(* Logix 5000 project; controller test vendor 1 type 14 code 151 rev 32.13; software revision 32.02; part 3 of 4 *)
(* tags used below, declared in another part *)
   _CopDes1 : DINT;
   _CopDes4 : DINT;
   _CopDes5 : DINT;
   _CopDes6 : DINT;
   _CopDes8 : DINT;
   _CopLength : DINT;
   _CopLength1 : DINT;
   _CopLength3 : DINT;
   _CopLength4 : DINT;
   _CopLength5 : DINT;
   _CopLength6 : DINT;
   _CopLength7 : DINT;
   _CopLength8 : DINT;
   _CopSource : DINT;
   _CopSource1 : DINT;
   _CopSource3 : DINT;
   _CopSource4 : DINT;
   _CopSource5 : DINT;
   _CopSource6 : DINT;
   _CopSource7 : DINT;
   _CopSource8 : DINT;
   _edbAoiFilterFlowAir : AOI_FilterSignal;
   _edbAoiFilterFlowO2 : AOI_FilterSignal;
   _edbAoiFilterPress : AOI_FilterSignal;
   _edbCanStore : BOOL;
   _edbFlowArrFiltered : REAL[1000,2];
   _edbFlowO2Filtered : REAL[1000,2];
   _edbHalfWindowFilterSize : DINT;
   _edbIdx : DINT;
   _edbParUseWeigths : BOOL;
   _edbParWeights : REAL[31];
   _edbPressArrFiltered : REAL[1000,2];
   _edbTypeOfFilter : DINT;
   _endPosition : DINT;
   _endPositionOld : DINT;
   _EndSendPosition : DINT;
   _i : DINT;
   _PointAfterEnd : DINT;
   _StartPointBerfore : DINT;
   _StartPosition : DINT;
   _StartpositionOld : DINT;
   AirConstantFlow : REAL;
   AirmADer : REAL;
   AirmAOut : REAL;
   AirmASlope : REAL;
   AirRampFlowIncreasePerAdjust : REAL;
   AirUp : CAM_PROFILE[1010];
   AnalogInputFlow : ALIAS FOR Local:2:I.Ch3Data;
   AnalogInputFlowAir : ALIAS FOR Local:2:I.Ch1Data;
   AnalogInputFlowO2 : ALIAS FOR Local:2:I.Ch0Data;
   AnalogInputPressure : ALIAS FOR Local:2:I.Ch2Data;
   AnalogOutFlowAir : ALIAS FOR Local:2:O.Ch1Data;
   AnalogOutFlowO2 : ALIAS FOR Local:2:O.Ch0Data;
   BreathDetect : BOOL;
   BreathDurationArr : REAL[50];   // 50 length array with seconds for each breath for calculation of minute avgVentStateArr. Calcualted from knowing meas at
   BreathDurationInMS : REAL;
   CalcNewData : BOOL;
   ConstansFlowNrCalc : REAL;
   ConstantFlowNrOfAdjustments : REAL;
   ConstantFlowTimeInMS : REAL;
   ConstantInspiratoryFlow : REAL;
   counter : DINT;   // Counter for Flow fill array
   CrsDynArr : REAL[50];   // 50 length array with dynamic respiraotry system compliance in ml/cmH2O, from measCalc()
   CrsQStatArr : REAL[50];   // 50 length array with quasistatic respiratory system compliance in ml/cmH2O, from measCalc()
   CsumData : DINT;
   CsumDataOld : DINT;
   data_changed : BOOL;
   endI : DINT;
   Exp : BOOL;
   expCount : INT;   // between 1-1000 to indicate where valveCtrl should read from expOpenCloseCtrl[]
   expCountLength : INT;   // between 1-1000 to indicate when valveCtrl should stop reading from expOpenCloseCtrl[], copied from nextExpCountLength by
   expCountlengthCalc : REAL;
   expCountLengthNew : REAL;
   expEndI : INT;
   expOpen : ALIAS FOR Local:1:O.Data.0;
   expOpenCloseCtrl : INT[1000];   // 1000 length array with open (1) or close (0) for exp valve, moved from nextexpOpenCloseCtrl[] by ISR_ValveCtrl()
   expOpenCloseCtrlNew : INT[1000];
   expStartI : INT;
   expTimeInMS : REAL;
   F1_pushed_new : BOOL;
   F1_pushed_old : BOOL;
   F2_pushed_new : BOOL;
   F2_pushed_old : BOOL;
   F3_pushed_new : BOOL;
   F3_pushed_old : BOOL;
   Fill : AOI_FillArrayReal;
   Fill50 : AOI_FillArrayReal50;
   Fillint : AOI_FillArrayInt;
   FillLoop : AOI_FillArray_Real2D;
   FiO2 : INT;   // 25-100%
   FiO2Running : INT;
   Floor : AOI_Floor;
   FlowAir : REAL[1000,2];   // 1000 length 2D FIFO array with flow values and status bits indicating if values have been analysed (1) or not (0) by mea
   FlowArrMem : REAL[1000,2];
   flowCalcOn : BOOL;
   FlowImaxArr : REAL[50];   // 50 length array with max insp flow in l/min, from measCalc()
   FlowO2 : REAL[1000,2];
   FlowO2Mem : REAL[1000,2];
   FractionAir : REAL;
   FractionO2 : REAL;
   GetSlaveValue : MOTION_INSTRUCTION;
   HMI_ScreenNo : DINT;
   HMIStart : BOOL;
   HMIStop : BOOL;
   i : DINT;
   I_E : STRING;   // part of I:E ratio: 1, 2, 3 or 4
   IE : STRING[4];
   IE_counter : DINT;
   IE_E : INT;
   IE_ERunning : INT;
   IE_I : INT;
   IE_IRunning : INT;
   Insp : BOOL;
   inspAirFlowCtrl : REAL[650];   // 650 length array with flow values for insp air valve, moved from nextInspAirFlowCtrl[] by ISR_ValveCtrl()
   inspAirFlowCtrlNew : REAL[650];
   inspCount : INT;   // between 1-650 to indicate where valveCtrl should read from inspAirFlowCtrl[] and inspO2FlowCtrl[]
   inspCountLength : INT;   // between 1-650 to indicate when valveCtrl should stop reading from inspAirFlowCtrl[] and inspO2FlowCtrl[], copied from ne
   inspCountLengthNew : REAL;
   inspCounts : REAL;
   InspiratoryRampTimeInMS : REAL;
   inspO2FlowCtrl : REAL[650];   // 650 length array with flow values for insp O2 valve, moved from nextInspO2FlowCtrl[] by ISR_ValveCtrl()
   inspO2FlowCtrlNew : REAL[650];
   inspPauseCalc : REAL;
   inspPauseNrOfAdjustments : REAL;
   inspPauseStartI : INT;
   inspPauseTime : INT;
   inspPauseTimeInMS : REAL;
   inspPauseTimePercent : REAL;
   inspPauseTimeRunning : INT;
   inspRampTime : INT;
   inspRampTimePercent : REAL;
   inspRampTimeRunning : INT;
   inspStartI : INT;
   inspTimeinMS : REAL;
   last_state : DINT;
   maxFlowAllowed : INT;
   message : STRING;
   Messages_to_user : STRING[10];
   Mode : STRING;
   MVArr : REAL[50];   // 50 length array with minute ventilation in l/min, from measCalc()
   NewExpOpenCloseAvail : BOOL;   // signal to valveCtrl to include new expOpenCloseCtrl[]to overwrite when expiration ended, set by calcBreath()
   newInspFlowAvil : BOOL;
   NewSettings : BOOL;
   NewTimeRate_p5 : DINT;
   NewTimeRate_p8 : DINT;
   nextExpCountLength : INT;   // between 1-1000 to indicate when valveCtrl should stop reading from expOpenCloseCtrl[], set by calcBreath()
   nextExpOpenCloseCtrl : INT[1000];   // 1000 length array with open (1) or close (0) for exp valve, set by calcBreath()
   nextInspAirFlowCtrl : REAL[650];   // 650 length array with flow values for insp air valve, set by calcBreath()
   nextInspCountLength : INT;   // between 1-650 to indicate when valveCtrl should stop reading from inspAirFlowCtrl[] and inspO2FlowCtrl[], set by calcBre
   nextInspO2FlowCtrl : REAL[650];   // 650 length array with flow values for insp O2 valve, set by calcBreath()
   O2 : DINT;
   O2ConstantFlow : REAL;
   O2mADer : REAL;
   O2mAOut : REAL;
   O2mASlope : REAL;
   O2RampFlowIncreasePerAdjust : REAL;
   O2Up : CAM_PROFILE[1010];

        [540].Status := 2, [541].Status := 2, [542].Status := 2, [543].Status := 2, [544].Status := 2, [545].Status := 2, [546].Status := 2, [547].Status := 2, [548].Status := 2, [549].Status := 2, [550].Status := 2, [551].Status := 2, [552].Status := 2, [553].Status := 2, [554].Status := 2, [555].Status := 2, [556].Status := 2, [557].Status := 2, [558].Status := 2, [559].Status := 2, [560].Status := 2, [561].Status := 2, [562].Status := 2, [563].Status := 2, [564].Status := 2, [565].Status := 2, [566].Status := 2, [567].Status := 2, [568].Status := 2, [569].Status := 2, [570].Status := 2, [571].Status := 2, [572].Status := 2, [573].Status := 2, [574].Status := 2, [575].Status := 2, [576].Status := 2, [577].Status := 2, [578].Status := 2, [579].Status := 2, [580].Status := 2, [581].Status := 2, [582].Status := 2, [583].Status := 2, [584].Status := 2, [585].Status := 2, [586].Status := 2, [587].Status := 2, [588].Status := 2, [589].Status := 2, [590].Status := 2, [591].Status := 2, [592].Status := 2, [593].Status := 2, [594].Status := 2, [595].Status := 2, [596].Status := 2, [597].Status := 2, [598].Status := 2, [599].Status := 2,
        [600].Status := 2, [601].Status := 2, [602].Status := 2, [603].Status := 2, [604].Status := 2, [605].Status := 2, [606].Status := 2, [607].Status := 2, [608].Status := 2, [609].Status := 2, [610].Status := 2, [611].Status := 2, [612].Status := 2, [613].Status := 2, [614].Status := 2, [615].Status := 2, [616].Status := 2, [617].Status := 2, [618].Status := 2, [619].Status := 2, [620].Status := 2, [621].Status := 2, [622].Status := 2, [623].Status := 2, [624].Status := 2, [625].Status := 2, [626].Status := 2, [627].Status := 2, [628].Status := 2, [629].Status := 2, [630].Status := 2, [631].Status := 2, [632].Status := 2, [633].Status := 2, [634].Status := 2, [635].Status := 2, [636].Status := 2, [637].Status := 2, [638].Status := 2, [639].Status := 2, [640].Status := 2, [641].Status := 2, [642].Status := 2, [643].Status := 2, [644].Status := 2, [645].Status := 2, [646].Status := 2, [647].Status := 2, [648].Status := 2, [649].Status := 2, [650].Status := 2, [651].Status := 2, [652].Status := 2, [653].Status := 2, [654].Status := 2, [655].Status := 2, [656].Status := 2, [657].Status := 2, [658].Status := 2, [659].Status := 2,
        [660].Status := 2, [661].Status := 2, [662].Status := 2, [663].Status := 2, [664].Status := 2, [665].Status := 2, [666].Status := 2, [667].Status := 2, [668].Status := 2, [669].Status := 2, [670].Status := 2, [671].Status := 2, [672].Status := 2, [673].Status := 2, [674].Status := 2, [675].Status := 2, [676].Status := 2, [677].Status := 2, [678].Status := 2, [679].Status := 2, [680].Status := 2, [681].Status := 2, [682].Status := 2, [683].Status := 2, [684].Status := 2, [685].Status := 2, [686].Status := 2, [687].Status := 2, [688].Status := 2, [689].Status := 2, [690].Status := 2, [691].Status := 2, [692].Status := 2, [693].Status := 2, [694].Status := 2, [695].Status := 2, [696].Status := 2, [697].Status := 2, [698].Status := 2, [699].Status := 2, [700].Status := 2, [701].Status := 2, [702].Status := 2, [703].Status := 2, [704].Status := 2, [705].Status := 2, [706].Status := 2, [707].Status := 2, [708].Status := 2, [709].Status := 2, [710].Status := 2, [711].Status := 2, [712].Status := 2, [713].Status := 2, [714].Status := 2, [715].Status := 2, [716].Status := 2, [717].Status := 2, [718].Status := 2, [719].Status := 2,
        [720].Status := 2, [721].Status := 2, [722].Status := 2, [723].Status := 2, [724].Status := 2, [725].Status := 2, [726].Status := 2, [727].Status := 2, [728].Status := 2, [729].Status := 2, [730].Status := 2, [731].Status := 2, [732].Status := 2, [733].Status := 2, [734].Status := 2, [735].Status := 2, [736].Status := 2, [737].Status := 2, [738].Status := 2, [739].Status := 2, [740].Status := 2, [741].Status := 2, [742].Status := 2, [743].Status := 2, [744].Status := 2, [745].Status := 2, [746].Status := 2, [747].Status := 2, [748].Status := 2, [749].Status := 2, [750].Status := 2, [751].Status := 2, [752].Status := 2, [753].Status := 2, [754].Status := 2, [755].Status := 2, [756].Status := 2, [757].Status := 2, [758].Status := 2, [759].Status := 2, [760].Status := 2, [761].Status := 2, [762].Status := 2, [763].Status := 2, [764].Status := 2, [765].Status := 2, [766].Status := 2, [767].Status := 2, [768].Status := 2, [769].Status := 2, [770].Status := 2, [771].Status := 2, [772].Status := 2, [773].Status := 2, [774].Status := 2, [775].Status := 2, [776].Status := 2, [777].Status := 2, [778].Status := 2, [779].Status := 2,
        [780].Status := 2, [781].Status := 2, [782].Status := 2, [783].Status := 2, [784].Status := 2, [785].Status := 2, [786].Status := 2, [787].Status := 2, [788].Status := 2, [789].Status := 2, [790].Status := 2, [791].Status := 2, [792].Status := 2, [793].Status := 2, [794].Status := 2, [795].Status := 2, [796].Status := 2, [797].Status := 2, [798].Status := 2, [799].Status := 2, [800].Status := 2, [801].Status := 2, [802].Status := 2, [803].Status := 2, [804].Status := 2, [805].Status := 2, [806].Status := 2, [807].Status := 2, [808].Status := 2, [809].Status := 2, [810].Status := 2, [811].Status := 2, [812].Status := 2, [813].Status := 2, [814].Status := 2, [815].Status := 2, [816].Status := 2, [817].Status := 2, [818].Status := 2, [819].Status := 2, [820].Status := 2, [821].Status := 2, [822].Status := 2, [823].Status := 2, [824].Status := 2, [825].Status := 2, [826].Status := 2, [827].Status := 2, [828].Status := 2, [829].Status := 2, [830].Status := 2, [831].Status := 2, [832].Status := 2, [833].Status := 2, [834].Status := 2, [835].Status := 2, [836].Status := 2, [837].Status := 2, [838].Status := 2, [839].Status := 2,
        [840].Status := 2, [841].Status := 2, [842].Status := 2, [843].Status := 2, [844].Status := 2, [845].Status := 2, [846].Status := 2, [847].Status := 2, [848].Status := 2, [849].Status := 2, [850].Status := 2, [851].Status := 2, [852].Status := 2, [853].Status := 2, [854].Status := 2, [855].Status := 2, [856].Status := 2, [857].Status := 2, [858].Status := 2, [859].Status := 2, [860].Status := 2, [861].Status := 2, [862].Status := 2, [863].Status := 2, [864].Status := 2, [865].Status := 2, [866].Status := 2, [867].Status := 2, [868].Status := 2, [869].Status := 2, [870].Status := 2, [871].Status := 2, [872].Status := 2, [873].Status := 2, [874].Status := 2, [875].Status := 2, [876].Status := 2, [877].Status := 2, [878].Status := 2, [879].Status := 2, [880].Status := 2, [881].Status := 2, [882].Status := 2, [883].Status := 2, [884].Status := 2, [885].Status := 2, [886].Status := 2, [887].Status := 2, [888].Status := 2, [889].Status := 2, [890].Status := 2, [891].Status := 2, [892].Status := 2, [893].Status := 2, [894].Status := 2, [895].Status := 2, [896].Status := 2, [897].Status := 2, [898].Status := 2, [899].Status := 2,
        [900].Status := 2, [901].Status := 2, [902].Status := 2, [903].Status := 2, [904].Status := 2, [905].Status := 2, [906].Status := 2, [907].Status := 2, [908].Status := 2, [909].Status := 2, [910].Status := 2, [911].Status := 2, [912].Status := 2, [913].Status := 2, [914].Status := 2, [915].Status := 2, [916].Status := 2, [917].Status := 2, [918].Status := 2, [919].Status := 2, [920].Status := 2, [921].Status := 2, [922].Status := 2, [923].Status := 2, [924].Status := 2, [925].Status := 2, [926].Status := 2, [927].Status := 2, [928].Status := 2, [929].Status := 2, [930].Status := 2, [931].Status := 2, [932].Status := 2, [933].Status := 2, [934].Status := 2, [935].Status := 2, [936].Status := 2, [937].Status := 2, [938].Status := 2, [939].Status := 2, [940].Status := 2, [941].Status := 2, [942].Status := 2, [943].Status := 2, [944].Status := 2, [945].Status := 2, [946].Status := 2, [947].Status := 2, [948].Status := 2, [949].Status := 2, [950].Status := 2, [951].Status := 2, [952].Status := 2, [953].Status := 2, [954].Status := 2, [955].Status := 2, [956].Status := 2, [957].Status := 2, [958].Status := 2, [959].Status := 2,
        [960].Status := 2, [961].Status := 2, [962].Status := 2, [963].Status := 2, [964].Status := 2, [965].Status := 2, [966].Status := 2, [967].Status := 2, [968].Status := 2, [969].Status := 2, [970].Status := 2, [971].Status := 2, [972].Status := 2, [973].Status := 2, [974].Status := 2, [975].Status := 2, [976].Status := 2, [977].Status := 2, [978].Status := 2, [979].Status := 2, [980].Status := 2, [981].Status := 2, [982].Status := 2, [983].Status := 2, [984].Status := 2, [985].Status := 2, [986].Status := 2, [987].Status := 2, [988].Status := 2, [989].Status := 2, [990].Status := 2, [991].Status := 2, [992].Status := 2, [993].Status := 2, [994].Status := 2, [995].Status := 2, [996].Status := 2, [997].Status := 2, [998].Status := 2, [999].Status := 2, [1000].Status := 2, [1001].Status := 2, [1002].Status := 2);
   PEEP : REAL := 4402.0;   // positive end expiratory pressure in cmH2O
   PEEPArr : REAL[50];   // 50 length array with positive end expiratory pressure in cmH2O, from measCalc()
   PEEPi : REAL;
   PEEPiArr : REAL[50];
   Ppeak : REAL := 10534.0;   // Ppeak
   PpeakArr : REAL[50];   // 50 length array with Ppeak from measCalc(), used for minAvg
   PpeakMaxValue : AOI_Max := (Out_Max := 10534.0, _i := 196);
   Pplat : REAL := 9761.556;   // plateau insp pressure in cmH2O
   PplatArr : REAL[50];   // 50 length array with plateau insp pressure in cmH2O, from measCalc()
   PplatBreathFrac : REAL := 0.2;
   PplatMean : AOI_Mean2D := (In_N0 := 186, In_N1 := 194, Out_Mean := 9761.556, _i := 195);
   PressArr : REAL[1000,2] := ([0,0] := 24.938433, [1,0] := 24.938433, [2,0] := 25.22523, [3,0] := 25.22523, [4,0] := 25.22523, [5,0] := 25.429173, [6,0] := 25.429173, [7,0] := 25.129631, [8,0] := 25.129631, [9,0] := 25.129631, [10,0] := 25.161495, [11,0] := 25.161495, [12,0] := 25.034033, [13,0] := 25.034033, [14,0] := 25.174244, [15,0] := 25.174244, [16,0] := 25.174244, [17,0] := 25.429173, [18,0] := 25.429173, [19,0] := 25.193363, [20,0] := 25.193363, [21,0] := 25.193363, [22,0] := 25.180616, [23,0] := 25.180616, [24,0] := 25.002167, [25,0] := 25.002167, [26,0] := 25.002167, [27,0] := 25.10414, [28,0] := 25.10414, [29,0] := 25.461039, [30,0] := 25.461039, [31,0] := 25.218855, [32,0] := 25.218855, [33,0] := 25.218855, [34,0] := 25.161495, [35,0] := 25.161495, [36,0] := 25.040407, [37,0] := 25.040407, [38,0] := 25.040407, [39,0] := 25.24435, [40,0] := 25.24435, [41,0] := 25.499277, [42,0] := 25.499277, [43,0] := 25.142378, [44,0] := 25.142378, [45,0] := 25.142378, [46,0] := 24.925688, [47,0] := 24.925688, [48,0] := 25.199736, [49,0] := 25.199736, [50,0] := 25.199736, [51,0] := 25.237976, [52,0] := 25.237976, [53,0] := 25.378187, [54,0] := 25.378187, [55,0] := 25.136003, [56,0] := 25.136003, [57,0] := 25.136003, [58,0] := 24.976673, [59,0] := 24.976673,
        [60,0] := 25.199736, [61,0] := 25.199736, [62,0] := 25.199736, [63,0] := 25.136003, [64,0] := 25.136003, [65,0] := 25.403679, [66,0] := 25.403679, [67,0] := 25.212482, [68,0] := 25.212482, [69,0] := 25.212482, [70,0] := 24.906569, [71,0] := 24.906569, [72,0] := 25.212482, [73,0] := 25.212482, [74,0] := 25.212482, [75,0] := 25.269842, [76,0] := 25.269842, [77,0] := 25.359066, [78,0] := 25.359066, [79,0] := 25.359066, [80,0] := 25.193363, [81,0] := 25.193363, [82,0] := 24.912941, [83,0] := 24.912941, [84,0] := 25.250723, [85,0] := 25.250723, [86,0] := 25.250723, [87,0] := 25.282587, [88,0] := 25.282587, [89,0] := 25.308083, [90,0] := 25.308083, [91,0] := 25.116884, [92,0] := 25.116884, [93,0] := 25.116884, [94,0] := 24.925688, [95,0] := 24.925688, [96,0] := 25.20611, [97,0] := 25.20611, [98,0] := 25.20611, [99,0] := 25.250723, [100,0] := 25.250723, [101,0] := 25.314455, [102,0] := 25.314455, [103,0] := 25.193363, [104,0] := 25.193363, [105,0] := 25.193363, [106,0] := 24.938433, [107,0] := 24.938433, [108,0] := 25.193363, [109,0] := 25.193363, [110,0] := 25.193363, [111,0] := 25.308083, [112,0] := 25.308083, [113,0] := 25.276215, [114,0] := 25.276215, [115,0] := 25.276215, [116,0] := 25.193363, [117,0] := 25.193363, [118,0] := 24.93206, [119,0] := 24.93206,
        [120,0] := 25.174244, [121,0] := 25.174244, [122,0] := 25.174244, [123,0] := 25.518398, [124,0] := 25.518398, [125,0] := 25.180616, [126,0] := 25.180616, [127,0] := 25.180616, [128,0] := 25.193363, [129,0] := 25.193363, [130,0] := 25.021286, [131,0] := 25.021286, [132,0] := 25.22523, [133,0] := 25.22523, [134,0] := 25.22523, [135,0] := 25.473785, [136,0] := 25.473785, [137,0] := 25.167871, [138,0] := 25.167871, [139,0] := 25.167871, [140,0] := 25.199736, [141,0] := 25.199736, [142,0] := 25.014912, [143,0] := 25.014912, [144,0] := 25.014912, [145,0] := 25.136003, [146,0] := 25.136003, [147,0] := 25.461039, [148,0] := 25.461039, [149,0] := 25.167871, [150,0] := 25.167871, [151,0] := 25.167871, [152,0] := 25.199736, [153,0] := 25.199736, [154,0] := 25.027658, [155,0] := 25.027658, [156,0] := 25.180616, [157,0] := 25.180616, [158,0] := 25.180616, [159,0] := 25.52477, [160,0] := 25.52477, [161,0] := 25.199736, [162,0] := 25.199736, [163,0] := 25.199736, [164,0] := 25.00854, [165,0] := 25.00854, [166,0] := 25.116884, [167,0] := 25.116884, [168,0] := 25.116884, [169,0] := 25.231602, [170,0] := 25.231602, [171,0] := 25.416426, [172,0] := 25.416426, [173,0] := 25.136003, [174,0] := 25.136003, [175,0] := 25.136003, [176,0] := 24.9703, [177,0] := 24.9703, [178,0] := 25.212482, [179,0] := 25.212482,
        [180,0] := 25.212482, [181,0] := 25.161495, [182,0] := 25.161495, [183,0] := 25.410053, [184,0] := 25.410053, [185,0] := 25.18699, [186,0] := 25.18699, [187,0] := 25.18699, [188,0] := 24.9703, [189,0] := 24.9703, [190,0] := 25.14875, [191,0] := 25.14875, [192,0] := 25.14875, [193,0] := 25.155123, [194,0] := 25.155123, [195,0] := 25.448294, [196,0] := 25.448294, [197,0] := 25.167871, [198,0] := 25.167871, [199,0] := 25.167871, [200,0] := 24.855581, [201,0] := 24.855581, [202,0] := 25.123259, [203,0] := 25.123259, [204,0] := 25.123259, [205,0] := 25.250723, [206,0] := 25.250723, [207,0] := 25.352694, [208,0] := 25.352694, [209,0] := 25.110512, [210,0] := 25.110512, [211,0] := 25.110512, [212,0] := 24.944807, [213,0] := 24.944807, [214,0] := 25.231602, [215,0] := 25.231602, [216,0] := 25.231602, [217,0] := 25.180616, [218,0] := 25.180616, [219,0] := 25.257095, [220,0] := 25.257095, [221,0] := 25.257095, [222,0] := 25.155123, [223,0] := 25.155123, [224,0] := 24.9703, [225,0] := 24.9703, [226,0] := 25.167871, [227,0] := 25.167871, [228,0] := 25.167871, [229,0] := 25.276215, [230,0] := 25.276215, [231,0] := 25.24435, [232,0] := 25.24435, [233,0] := 25.199736, [234,0] := 25.199736, [235,0] := 25.199736, [236,0] := 24.855581, [237,0] := 24.855581, [238,0] := 25.167871, [239,0] := 25.167871,
        [240,0] := 25.167871, [241,0] := 25.38456, [242,0] := 25.38456, [243,0] := 25.250723, [244,0] := 25.250723, [245,0] := 25.250723, [246,0] := 25.155123, [247,0] := 25.155123, [248,0] := 24.900196, [249,0] := 24.900196, [250,0] := 25.237976, [251,0] := 25.237976, [252,0] := 25.237976, [253,0] := 25.461039, [254,0] := 25.461039, [255,0] := 25.193363, [256,0] := 25.193363, [257,0] := 25.193363, [258,0] := 25.199736, [259,0] := 25.199736, [260,0] := 25.00854, [261,0] := 25.00854, [262,0] := 25.237976, [263,0] := 25.237976, [264,0] := 25.237976, [265,0] := 25.422798, [266,0] := 25.422798, [267,0] := 25.193363, [268,0] := 25.193363, [269,0] := 25.193363, [270,0] := 25.18699, [271,0] := 25.18699, [272,0] := 25.065899, [273,0] := 25.065899, [274,0] := 25.155123, [275,0] := 25.155123, [276,0] := 25.155123, [277,0] := 25.473785, [278,0] := 25.473785, [279,0] := 25.20611, [280,0] := 25.20611, [281,0] := 25.20611, [282,0] := 24.98942, [283,0] := 24.98942, [284,0] := 25.142378, [285,0] := 25.142378, [286,0] := 25.142378, [287,0] := 25.250723, [288,0] := 25.250723, [289,0] := 25.48653, [290,0] := 25.48653, [291,0] := 25.142378, [292,0] := 25.142378, [293,0] := 25.142378, [294,0] := 24.893822, [295,0] := 24.893822, [296,0] := 25.199736, [297,0] := 25.199736, [298,0] := 25.199736, [299,0] := 25.193363,
        [300,0] := 25.193363, [301,0] := 25.295334, [302,0] := 25.295334, [303,0] := 25.199736, [304,0] := 25.199736, [305,0] := 25.199736, [306,0] := 24.944807, [307,0] := 24.944807, [308,0] := 25.193363, [309,0] := 25.193363, [310,0] := 25.193363, [311,0] := 25.212482, [312,0] := 25.212482, [313,0] := 25.371813, [314,0] := 25.371813, [315,0] := 25.371813, [316,0] := 25.250723, [317,0] := 25.250723, [318,0] := 24.8747, [319,0] := 24.8747, [320,0] := 25.167871, [321,0] := 25.167871, [322,0] := 25.167871, [323,0] := 25.269842, [324,0] := 25.269842, [325,0] := 25.36544, [326,0] := 25.36544, [327,0] := 25.180616, [328,0] := 25.180616, [329,0] := 25.180616, [330,0] := 24.849209, [331,0] := 24.849209, [332,0] := 25.199736, [333,0] := 25.199736, [334,0] := 25.199736, [335,0] := 25.333574, [336,0] := 25.333574, [337,0] := 25.250723, [338,0] := 25.250723, [339,0] := 25.250723, [340,0] := 25.123259, [341,0] := 25.123259, [342,0] := 24.893822, [343,0] := 24.893822, [344,0] := 25.22523, [345,0] := 25.22523, [346,0] := 25.22523, [347,0] := 25.346321, [348,0] := 25.346321, [349,0] := 25.199736, [350,0] := 25.199736, [351,0] := 25.199736, [352,0] := 25.212482, [353,0] := 25.212482, [354,0] := 25.002167, [355,0] := 25.002167, [356,0] := 25.212482, [357,0] := 25.212482, [358,0] := 25.212482, [359,0] := 25.480158,
        [360,0] := 25.480158, [361,0] := 25.24435, [362,0] := 25.24435, [363,0] := 25.24435, [364,0] := 25.161495, [365,0] := 25.161495, [366,0] := 25.014912, [367,0] := 25.014912, [368,0] := 25.218855, [369,0] := 25.218855, [370,0] := 25.218855, [371,0] := 25.52477, [372,0] := 25.52477, [373,0] := 25.218855, [374,0] := 25.218855, [375,0] := 25.218855, [376,0] := 25.167871, [377,0] := 25.167871, [378,0] := 25.065899, [379,0] := 25.065899, [380,0] := 25.257095, [381,0] := 25.257095, [382,0] := 25.257095, [383,0] := 25.441917, [384,0] := 25.441917, [385,0] := 25.110512, [386,0] := 25.110512, [387,0] := 25.110512, [388,0] := 25.161495, [389,0] := 25.161495, [390,0] := 25.123259, [391,0] := 25.123259, [392,0] := 25.123259, [393,0] := 25.14875, [394,0] := 25.14875, [395,0] := 25.422798, [396,0] := 25.422798, [397,0] := 25.22523, [398,0] := 25.22523, [399,0] := 25.22523, [400,0] := 24.963928, [401,0] := 24.963928, [402,0] := 25.10414, [403,0] := 25.10414, [404,0] := 25.10414, [405,0] := 25.174244, [406,0] := 25.174244, [407,0] := 25.461039, [408,0] := 25.461039, [409,0] := 25.167871, [410,0] := 25.167871, [411,0] := 25.167871, [412,0] := 24.881075, [413,0] := 24.881075, [414,0] := 25.237976, [415,0] := 25.237976, [416,0] := 25.237976, [417,0] := 25.218855, [418,0] := 25.218855, [419,0] := 25.397306,
        [420,0] := 25.397306, [421,0] := 25.078644, [422,0] := 25.078644, [423,0] := 25.078644, [424,0] := 24.912941, [425,0] := 24.912941, [426,0] := 25.218855, [427,0] := 25.218855, [428,0] := 25.218855, [429,0] := 25.142378, [430,0] := 25.142378, [431,0] := 25.327202, [432,0] := 25.327202, [433,0] := 25.180616, [434,0] := 25.180616, [435,0] := 25.180616, [436,0] := 24.93206, [437,0] := 24.93206, [438,0] := 25.212482, [439,0] := 25.212482, [440,0] := 25.212482, [441,0] := 25.167871, [442,0] := 25.167871, [443,0] := 25.339947, [444,0] := 25.339947, [445,0] := 25.339947, [446,0] := 25.18699, [447,0] := 25.18699, [448,0] := 24.868328, [449,0] := 24.868328, [450,0] := 25.20611, [451,0] := 25.20611, [452,0] := 25.20611, [453,0] := 25.250723, [454,0] := 25.250723, [455,0] := 25.320827, [456,0] := 25.320827, [457,0] := 25.155123, [458,0] := 25.155123, [459,0] := 25.155123, [460,0] := 24.900196, [461,0] := 24.900196, [462,0] := 25.237976, [463,0] := 25.237976, [464,0] := 25.237976, [465,0] := 25.327202, [466,0] := 25.327202, [467,0] := 25.20611, [468,0] := 25.20611, [469,0] := 25.20611, [470,0] := 25.20611, [471,0] := 25.20611, [472,0] := 24.944807, [473,0] := 24.944807, [474,0] := 25.218855, [475,0] := 25.218855, [476,0] := 25.218855, [477,0] := 25.410053, [478,0] := 25.410053, [479,0] := 25.237976,
        [480,0] := 25.237976, [481,0] := 25.237976, [482,0] := 25.257095, [483,0] := 25.257095, [484,0] := 24.98942, [485,0] := 24.98942, [486,0] := 25.231602, [487,0] := 25.231602, [488,0] := 25.231602, [489,0] := 25.480158, [490,0] := 25.480158, [491,0] := 25.282587, [492,0] := 25.282587, [493,0] := 25.282587, [494,0] := 25.180616, [495,0] := 25.180616, [496,0] := 25.014912, [497,0] := 25.014912, [498,0] := 25.218855, [499,0] := 25.218855, [500,0] := 25.218855, [501,0] := 25.492905, [502,0] := 25.492905, [503,0] := 25.14875, [504,0] := 25.14875, [505,0] := 25.14875, [506,0] := 25.09139, [507,0] := 25.09139, [508,0] := 25.034033, [509,0] := 25.034033, [510,0] := 25.034033, [511,0] := 25.22523, [512,0] := 25.22523, [513,0] := 25.473785, [514,0] := 25.473785, [515,0] := 25.078644, [516,0] := 25.078644, [517,0] := 25.078644, [518,0] := 25.18699, [519,0] := 25.18699, [520,0] := 25.040407, [521,0] := 25.040407, [522,0] := 25.155123, [523,0] := 25.155123, [524,0] := 25.155123, [525,0] := 25.441917, [526,0] := 25.441917, [527,0] := 25.18699, [528,0] := 25.18699, [529,0] := 25.18699, [530,0] := 25.167871, [531,0] := 25.167871, [532,0] := 25.059525, [533,0] := 25.059525, [534,0] := 25.167871, [535,0] := 25.167871, [536,0] := 25.167871, [537,0] := 25.480158, [538,0] := 25.480158, [539,0] := 25.231602,
        [540,0] := 25.231602, [541,0] := 25.231602, [542,0] := 25.04678, [543,0] := 25.04678, [544,0] := 25.09139, [545,0] := 25.09139, [546,0] := 25.09139, [547,0] := 25.231602, [548,0] := 25.231602, [549,0] := 25.499277, [550,0] := 25.499277, [551,0] := 25.155123, [552,0] := 25.155123, [553,0] := 25.155123, [554,0] := 24.98942, [555,0] := 24.98942, [556,0] := 25.136003, [557,0] := 25.136003, [558,0] := 25.212482, [559,0] := 25.212482, [560,0] := 25.212482, [561,0] := 25.378187, [562,0] := 25.378187, [563,0] := 25.193363, [564,0] := 25.193363, [565,0] := 25.193363, [566,0] := 24.995792, [567,0] := 24.995792, [568,0] := 25.155123, [569,0] := 25.155123, [570,0] := 25.142378, [571,0] := 25.142378, [572,0] := 25.142378, [573,0] := 25.378187, [574,0] := 25.378187, [575,0] := 25.18699, [576,0] := 25.18699, [577,0] := 25.18699, [578,0] := 24.938433, [579,0] := 24.938433, [580,0] := 25.161495, [581,0] := 25.161495, [582,0] := 25.161495, [583,0] := 25.129631, [584,0] := 25.129631, [585,0] := 25.435545, [586,0] := 25.435545, [587,0] := 25.231602, [588,0] := 25.231602, [589,0] := 25.231602, [590,0] := 24.861956, [591,0] := 24.861956, [592,0] := 25.155123, [593,0] := 25.155123, [594,0] := 25.155123, [595,0] := 25.237976, [596,0] := 25.237976, [597,0] := 25.339947, [598,0] := 25.339947, [599,0] := 25.339947,
        [600,0] := 25.174244, [601,0] := 25.174244, [602,0] := 24.938433, [603,0] := 24.938433, [604,0] := 25.18699, [605,0] := 25.18699, [606,0] := 25.18699, [607,0] := 25.24435, [608,0] := 25.24435, [609,0] := 25.180616, [610,0] := 25.180616, [611,0] := 25.180616, [612,0] := 25.180616, [613,0] := 25.180616, [614,0] := 24.912941, [615,0] := 24.912941, [616,0] := 25.174244, [617,0] := 25.174244, [618,0] := 25.174244, [619,0] := 25.346321, [620,0] := 25.346321, [621,0] := 25.237976, [622,0] := 25.237976, [623,0] := 25.237976, [624,0] := 25.199736, [625,0] := 25.199736, [626,0] := 24.8747, [627,0] := 24.8747, [628,0] := 25.212482, [629,0] := 25.212482, [630,0] := 25.212482, [631,0] := 25.492905, [632,0] := 25.492905, [633,0] := 25.129631, [634,0] := 25.129631, [635,0] := 25.129631, [636,0] := 25.09139, [637,0] := 25.09139, [638,0] := 25.065899, [639,0] := 25.065899, [640,0] := 25.180616, [641,0] := 25.180616, [642,0] := 25.180616, [643,0] := 25.435545, [644,0] := 25.435545, [645,0] := 25.142378, [646,0] := 25.142378, [647,0] := 25.142378, [648,0] := 25.155123, [649,0] := 25.155123, [650,0] := 25.04678, [651,0] := 25.04678, [652,0] := 25.174244, [653,0] := 25.174244, [654,0] := 25.174244, [655,0] := 25.441917, [656,0] := 25.441917, [657,0] := 25.20611, [658,0] := 25.20611, [659,0] := 25.20611,
        [660,0] := 25.04678, [661,0] := 25.04678, [662,0] := 25.072271, [663,0] := 25.072271, [664,0] := 25.237976, [665,0] := 25.237976, [666,0] := 25.237976, [667,0] := 25.467413, [668,0] := 25.467413, [669,0] := 25.231602, [670,0] := 25.231602, [671,0] := 25.231602, [672,0] := 24.963928, [673,0] := 24.963928, [674,0] := 25.167871, [675,0] := 25.167871, [676,0] := 25.167871, [677,0] := 25.212482, [678,0] := 25.212482, [679,0] := 25.397306, [680,0] := 25.397306, [681,0] := 25.072271, [682,0] := 25.072271, [683,0] := 25.072271, [684,0] := 24.925688, [685,0] := 24.925688, [686,0] := 25.22523, [687,0] := 25.22523, [688,0] := 25.22523, [689,0] := 25.18699, [690,0] := 25.18699, [691,0] := 25.378187, [692,0] := 25.378187, [693,0] := 25.180616, [694,0] := 25.180616, [695,0] := 25.180616, [696,0] := 24.957552, [697,0] := 24.957552, [698,0] := 25.199736, [699,0] := 25.199736, [700,0] := 25.199736, [701,0] := 25.161495, [702,0] := 25.161495, [703,0] := 25.36544, [704,0] := 25.36544, [705,0] := 25.257095, [706,0] := 25.257095, [707,0] := 25.257095, [708,0] := 24.8747, [709,0] := 24.8747, [710,0] := 25.142378, [711,0] := 25.142378, [712,0] := 25.142378, [713,0] := 25.237976, [714,0] := 25.237976, [715,0] := 25.327202, [716,0] := 25.327202, [717,0] := 25.327202, [718,0] := 25.155123, [719,0] := 25.155123,
        [720,0] := 24.893822, [721,0] := 24.893822, [722,0] := 25.20611, [723,0] := 25.20611, [724,0] := 25.20611, [725,0] := 25.390934, [726,0] := 25.390934, [727,0] := 25.18699, [728,0] := 25.18699, [729,0] := 25.18699, [730,0] := 25.174244, [731,0] := 25.174244, [732,0] := 24.944807, [733,0] := 24.944807, [734,0] := 25.231602, [735,0] := 25.231602, [736,0] := 25.231602, [737,0] := 25.461039, [738,0] := 25.461039, [739,0] := 25.269842, [740,0] := 25.269842, [741,0] := 25.269842, [742,0] := 25.212482, [743,0] := 25.212482, [744,0] := 24.9703, [745,0] := 24.9703, [746,0] := 25.136003, [747,0] := 25.136003, [748,0] := 25.136003, [749,0] := 25.52477, [750,0] := 25.52477, [751,0] := 25.218855, [752,0] := 25.218855, [753,0] := 25.218855, [754,0] := 25.129631, [755,0] := 25.129631, [756,0] := 24.983047, [757,0] := 24.983047, [758,0] := 25.193363, [759,0] := 25.193363, [760,0] := 25.193363, [761,0] := 25.52477, [762,0] := 25.52477, [763,0] := 25.142378, [764,0] := 25.142378, [765,0] := 25.142378, [766,0] := 25.097763, [767,0] := 25.097763, [768,0] := 25.110512, [769,0] := 25.110512, [770,0] := 25.237976, [771,0] := 25.237976, [772,0] := 25.237976, [773,0] := 25.467413, [774,0] := 25.467413, [775,0] := 25.155123, [776,0] := 25.155123, [777,0] := 25.155123, [778,0] := 25.136003, [779,0] := 25.136003,
        [780,0] := 25.161495, [781,0] := 25.161495, [782,0] := 25.22523, [783,0] := 25.22523, [784,0] := 25.22523, [785,0] := 25.448294, [786,0] := 25.448294, [787,0] := 25.20611, [788,0] := 25.20611, [789,0] := 25.20611, [790,0] := 25.04678, [791,0] := 25.04678, [792,0] := 25.116884, [793,0] := 25.116884, [794,0] := 25.116884, [795,0] := 25.218855, [796,0] := 25.218855, [797,0] := 25.480158, [798,0] := 25.480158, [799,0] := 25.136003, [800,0] := 25.136003, [801,0] := 25.136003, [802,0] := 24.893822, [803,0] := 24.893822, [804,0] := 25.212482, [805,0] := 25.212482, [806,0] := 25.212482, [807,0] := 25.237976, [808,0] := 25.237976, [809,0] := 25.38456, [810,0] := 25.38456, [811,0] := 25.167871, [812,0] := 25.167871, [813,0] := 25.167871, [814,0] := 24.912941, [815,0] := 24.912941, [816,0] := 25.237976, [817,0] := 25.237976, [818,0] := 25.237976, [819,0] := 25.193363, [820,0] := 25.193363, [821,0] := 25.320827, [822,0] := 25.320827, [823,0] := 25.212482, [824,0] := 25.212482, [825,0] := 25.212482, [826,0] := 24.919315, [827,0] := 24.919315, [828,0] := 25.161495, [829,0] := 25.161495, [830,0] := 25.161495, [831,0] := 25.339947, [832,0] := 25.339947, [833,0] := 25.320827, [834,0] := 25.320827, [835,0] := 25.320827, [836,0] := 25.142378, [837,0] := 25.142378, [838,0] := 24.957552, [839,0] := 24.957552,
        [840,0] := 25.237976, [841,0] := 25.237976, [842,0] := 25.237976, [843,0] := 25.390934, [844,0] := 25.390934, [845,0] := 25.231602, [846,0] := 25.231602, [847,0] := 25.231602, [848,0] := 25.237976, [849,0] := 25.237976, [850,0] := 24.925688, [851,0] := 24.925688, [852,0] := 25.22523, [853,0] := 25.22523, [854,0] := 25.22523, [855,0] := 25.461039, [856,0] := 25.461039, [857,0] := 25.167871, [858,0] := 25.167871, [859,0] := 25.167871, [860,0] := 25.20611, [861,0] := 25.20611, [862,0] := 25.014912, [863,0] := 25.014912, [864,0] := 25.014912, [865,0] := 25.193363, [866,0] := 25.193363, [867,0] := 25.473785, [868,0] := 25.473785, [869,0] := 25.250723, [870,0] := 25.250723, [871,0] := 25.250723, [872,0] := 25.161495, [873,0] := 25.161495, [874,0] := 24.976673, [875,0] := 24.976673, [876,0] := 25.26347, [877,0] := 25.26347, [878,0] := 25.20611, [879,0] := 25.20611, [880,0] := 25.20611, [881,0] := 24.957552, [882,0] := 24.957552, [883,0] := 25.212482, [884,0] := 25.212482, [885,0] := 25.212482, [886,0] := 25.320827, [887,0] := 25.320827, [888,0] := 25.250723, [889,0] := 25.250723, [890,0] := 25.250723, [891,0] := 25.193363, [892,0] := 25.193363, [893,0] := 24.98942, [894,0] := 24.98942, [895,0] := 25.20611, [896,0] := 25.20611, [897,0] := 25.20611, [898,0] := 25.454666, [899,0] := 25.454666,
        [900,0] := 25.231602, [901,0] := 25.231602, [902,0] := 25.231602, [903,0] := 25.161495, [904,0] := 25.161495, [905,0] := 24.983047, [906,0] := 24.983047, [907,0] := 25.20611, [908,0] := 25.20611, [909,0] := 25.20611, [910,0] := 25.537518, [911,0] := 25.537518, [912,0] := 25.129631, [913,0] := 25.129631, [914,0] := 25.129631, [915,0] := 25.180616, [916,0] := 25.180616, [917,0] := 24.98942, [918,0] := 24.98942, [919,0] := 24.98942, [920,0] := 25.269842, [921,0] := 25.269842, [922,0] := 25.492905, [923,0] := 25.492905, [924,0] := 25.199736, [925,0] := 25.199736, [926,0] := 25.199736, [927,0] := 25.14875, [928,0] := 25.14875, [929,0] := 25.110512, [930,0] := 25.110512, [931,0] := 25.110512, [932,0] := 25.167871, [933,0] := 25.167871, [934,0] := 25.378187, [935,0] := 25.378187, [936,0] := 25.218855, [937,0] := 25.218855, [938,0] := 25.218855, [939,0] := 25.078644, [940,0] := 25.078644, [941,0] := 25.097763, [942,0] := 25.097763, [943,0] := 25.097763, [944,0] := 25.129631, [945,0] := 25.129631, [946,0] := 25.50565, [947,0] := 25.50565, [948,0] := 25.161495, [949,0] := 25.161495, [950,0] := 25.161495, [951,0] := 24.98942, [952,0] := 24.98942, [953,0] := 25.199736, [954,0] := 25.199736, [955,0] := 25.199736, [956,0] := 25.20611, [957,0] := 25.20611, [958,0] := 25.429173, [959,0] := 25.429173,
        [960,0] := 25.116884, [961,0] := 25.116884, [962,0] := 25.116884, [963,0] := 24.925688, [964,0] := 24.925688, [965,0] := 25.180616, [966,0] := 25.180616, [967,0] := 25.180616, [968,0] := 25.180616, [969,0] := 25.180616, [970,0] := 25.231602, [971,0] := 25.231602, [972,0] := 25.180616, [973,0] := 25.180616, [974,0] := 25.180616, [975,0] := 24.9703, [976,0] := 24.9703, [977,0] := 25.20611, [978,0] := 25.20611, [979,0] := 25.20611, [980,0] := 25.333574, [981,0] := 25.333574, [982,0] := 25.295334, [983,0] := 25.295334, [984,0] := 25.231602, [985,0] := 25.231602, [986,0] := 25.231602, [987,0] := 24.881075, [988,0] := 24.881075, [989,0] := 25.193363, [990,0] := 25.193363, [991,0] := 25.193363, [992,0] := 25.480158, [993,0] := 25.480158, [994,0] := 25.193363, [995,0] := 25.193363, [996,0] := 25.193363, [997,0] := 25.174244, [998,0] := 25.174244);   // 1000 length 2D FIFO array with pressure values and status bits indicating if values have been analysed (1) or not (0) by measCalc()
   PressArrMem : REAL[1000,2];
   PressHtreshold : ALIAS FOR Local:2:C.Ch2HAlarmLimit;
   Pressure : REAL := -0.28125;
   pressWDAlertCount : INT;   // between 1-5 to close valve for 5x0.01 s=0.05 sec when press too high
   PressWDAlertMax : DINT;
   RampNrCalc : REAL := 20.000002;
   RampNrOfAdjustments : REAL := 20.0;
   RampTime : REAL[650] := ([0] := -10.0, [2] := 10.0, [3] := 20.0, [4] := 30.0, [5] := 40.0, [6] := 50.0, [7] := 60.0, [8] := 70.0, [9] := 80.0, [10] := 90.0, [11] := 100.0, [12] := 110.0, [13] := 120.0, [14] := 130.0, [15] := 140.0, [16] := 150.0, [17] := 160.0, [18] := 170.0, [19] := 180.0, [20] := 190.0, [21] := 200.0, [22] := 210.0, [23] := 220.0, [24] := 230.0, [25] := 240.0, [26] := 250.0, [27] := 260.0, [28] := 270.0, [29] := 280.0, [30] := 290.0, [31] := 300.0, [32] := 310.0, [33] := 320.0, [34] := 330.0, [35] := 340.0, [36] := 350.0, [37] := 360.0, [38] := 370.0, [39] := 380.0, [40] := 390.0, [41] := 400.0, [42] := 410.0, [43] := 420.0, [44] := 430.0, [45] := 440.0, [46] := 450.0, [47] := 460.0, [48] := 470.0, [49] := 480.0, [50] := 490.0, [51] := 500.0, [52] := 510.0, [53] := 520.0, [54] := 530.0, [55] := 540.0, [56] := 550.0, [57] := 560.0, [58] := 570.0, [59] := 580.0, [60] := 590.0,
        [61] := 600.0, [62] := 610.0, [63] := 620.0, [64] := 630.0, [65] := 640.0, [66] := 650.0, [67] := 660.0, [68] := 670.0, [69] := 680.0, [70] := 690.0, [71] := 700.0, [72] := 710.0, [73] := 720.0, [74] := 730.0, [75] := 740.0, [76] := 750.0, [77] := 760.0, [78] := 770.0, [79] := 780.0, [80] := 790.0, [81] := 800.0, [82] := 810.0, [83] := 820.0, [84] := 830.0, [85] := 840.0, [86] := 850.0, [87] := 860.0, [88] := 870.0, [89] := 880.0, [90] := 890.0);
   Raw : REAL := 2.440968;   // airway resistance in cmH2O/l/s
   RawArr : REAL[50];   // 50 length array with airway resistance in cmH2O/l/s
   Round : AOI_Round := (In_X := 8.2);
   RR : REAL := 15.0;   // respiratory rate in 1/min
   RRArr : REAL[50];   // 50 length array with respiratory rate in 1/min, from measCalc()
   RRate : INT := 15;
   RRateRunning : INT := 15;
   RRin : INT;   // 6-40 1/min
   RunModes : STRING[4] := ([0] := 'VC');
   SampelRateChangeAllowed : BOOL;
   Samplerate : DINT := 100;   // The rate in Hz that samples is collected
   Samplerate_Old : DINT;
   SetupDone : BOOL := 1;
   SetupState : DINT;
   Start_Stop : BOOL;
   StartPoint : INT := 186;
   StartPointMean : REAL := 8.0;
   StartPointValue : REAL := 8.2;
   StartSendPosition : DINT := -30;
   StartVent : BOOL;   // 1: start ventilating patient, 0: do nothing
   state : DINT := 3;
   state0 : BOOL;
   state1 : BOOL;
   state2 : BOOL;
   state3 : BOOL;
   state_selected : BOOL;
   StateBreathDetect : DINT;
   StateCalcBreath : DINT;
   StateInitVent : DINT;
   StateMain : DINT := 20;
   StatemeasCalc : DINT;
   StateValveCtrl : DINT;
   StopVent : BOOL;   // 1: stop ventilating patient after finished breath, shut down not necessary ISRs
   testtag : DINT := 13287;
   Time : DINT := 4800;
   Timer : DINT;
   TimeRate : DINT := 10000;
   TimerDone : BOOL;
   tipause : INT := 250;
   tmp_value : DINT;
   totalCount : REAL := 400.00003;
   totTime : INT;
   TrendAirFlow : REAL;
   TrendO2Flow : REAL;
   trigger : BOOL;
   valveUpdInterval : REAL := 10.0;
   VentOn : BOOL;   // 1: keep ventilatin patient, checked by ISR_ValveCtrl() to stop after breath and measCalc()
   ventState : INT;   // 0: stopped, 1: insp, 2: inspPause, 3: exp, 4: expPause
   VentStateArr : INT[1000];   // 1000 length array with ventilator state at each flow and pressure reading, used for calculation
   Vt : INT := 600;   // 200-600 ml
   Vti : REAL := 3201.7312;   // insp tidal volume in ml
   VtiArr : REAL[50];   // 50 length array with insp tidal volume in ml, from measCalc()
   VtRunning : INT := 600;
END_VAR

PROGRAM BreathDetect   (* main routine Main *)

ROUTINE Main   (* structured text *)
   
END_ROUTINE
END_PROGRAM

PROGRAM calcBreath   (* main routine Main *)

ROUTINE Main   (* structured text *)
   //Saves o2 and air inspiratory flows in l/min as 100 Hz arrays for ISR_valveCtrl() to
   //read and convert to a current securing these defined flows delivered to
   //the patient.
   
   if StateCalcBreath = 10 then;
   
   	//Calculate durations
   	inspPauseTimePercent := inspPauseTime/100; 	//Percentage of whole inspIE_In where there is a pause (in the end)
   	inspRampTimePercent := inspRampTime/100; 	//Percentage of active inspIE_In (when there is flow)
   	BreathDurationInMS := (1/RRate) * 60000;
   	inspTimeinMS := IE_I * (BreathDurationInMS/(IE_I+IE_E));
   	totalCount := BreathDurationInMS/valveUpdInterval;
   	inspCounts := inspTimeinMS/valveUpdInterval;
   	AOI_Floor(Floor,inspCounts,inspCountLengthNew);
   	expTimeInMS := BreathDurationInMS - inspTimeinMS;
   	expCountlengthCalc := totalCount-inspCountLengthNew;
   	AOI_Floor(Floor, expCountlengthCalc, expCountLengthNew);
   
   	//Calculate part of inspIE_In where valves are open
   	inspPauseTimeInMS := inspPauseTimePercent * BreathDurationInMS;
   	InspiratoryRampTimeInMS := inspRampTimePercent * BreathDurationInMS;
   	ConstantFlowTimeInMS := inspTimeinMS - inspPauseTimeInMS - InspiratoryRampTimeInMS;
   
   
   	//Calculate flow in L/min required to reach Vt in active inspIE_In
   	//(assuming a linear ramp)
   	ConstantInspiratoryFlow := 1/(ConstantFlowTimeInMS+0.5*InspiratoryRampTimeInMS)*Vt*60;
   
   	//This needs to be warned to the user - We will need a handle in HMI to not
   	//allow such settings if we are stuck with this limit on max flow
   	if ConstantInspiratoryFlow > maxFlowAllowed then;
   	    COP(Messages_to_user[2], message, 82);
   	end_if;
   
   	//Calculate split between O2 and Air
   	FractionAir := ((1-FiO2/100)/0.79);
   	FractionO2 := 1 - FractionAir;
   
   	//Calculate Ramp samples for O2 and Air
   	O2ConstantFlow := FractionO2 * ConstantInspiratoryFlow; 		//L/min
   	AirConstantFlow := FractionAir * ConstantInspiratoryFlow; 		//L/min
   
   	RampNrCalc := InspiratoryRampTimeInMS/valveUpdInterval;
   	AOI_Floor(Floor, RampNrCalc,RampNrOfAdjustments);
   	O2RampFlowIncreasePerAdjust := O2ConstantFlow/RampNrOfAdjustments;
   	AirRampFlowIncreasePerAdjust := AirConstantFlow/RampNrOfAdjustments;
   
   	ConstansFlowNrCalc := ConstantFlowTimeInMS/valveUpdInterval;
   	AOI_Floor(Floor, ConstansFlowNrCalc,ConstantFlowNrOfAdjustments );
   	inspPauseCalc := inspPauseTimeInMS/valveUpdInterval;
   	AOI_Floor(Floor, inspPauseCalc,inspPauseNrOfAdjustments );
   
   	//Build control arrays
   	AOI_FillArrayReal(Fill, inspO2FlowCtrlNew, 0, 650);
   	AOI_FillArrayReal(Fill, inspAirFlowCtrlNew, 0, 650);
   	AOI_FillArrayInt(Fillint, expOpenCloseCtrlNew, 0, 1000);
   
   	//inspiratory
   	for i :=0 to inspCountLengthNew by 1 do;
   	    if i <= RampNrOfAdjustments then;
   	        RampTime[i] := valveUpdInterval*(i-1);
   	        inspO2FlowCtrlNew[i] := i *  O2RampFlowIncreasePerAdjust;
   	        inspAirFlowCtrlNew[i] := i *  AirRampFlowIncreasePerAdjust;
   	    elsif i > RampNrOfAdjustments and i < RampNrOfAdjustments+ConstantFlowNrOfAdjustments then;
   	        inspO2FlowCtrlNew[i] := O2ConstantFlow;
   	        inspAirFlowCtrlNew[i] := AirConstantFlow;
   	    elsif i > (RampNrOfAdjustments+ConstantFlowNrOfAdjustments) and i <= (RampNrOfAdjustments+ConstantFlowNrOfAdjustments+inspPauseNrOfAdjustments) then;
   	        inspO2FlowCtrlNew[i] := 0;
   	        inspAirFlowCtrlNew[i] := 0;
   	    end_if;
   	end_for;
   
   	//expiratory
   	AOI_FillArrayInt(Fillint, expOpenCloseCtrlNew, 1, expCountLengthNew);
   
   	// Copy calculated data for Inspiratoty to next breath cycles
   	COP(inspO2FlowCtrlNew[0], nextInspO2FlowCtrl[0], 650);
   	COP(inspAirFlowCtrlNew[0], nextInspAirFlowCtrl[0], 650);
   	nextInspCountLength := inspCountLengthNew;
   
   	// Copy calculated data for Expiratory to next breath cycles
   	COP(expOpenCloseCtrlNew[0], nextExpOpenCloseCtrl[0], 1000);
   	nextExpCountLength := expCountLengthNew;
   
   	NewSettings := 0;
   	newInspFlowAvil := 1;
   	NewExpOpenCloseAvail:= 1;
   	StateCalcBreath := 0;
   
   end_if;
   
   
END_ROUTINE
END_PROGRAM

PROGRAM GUI   (* main routine Handle_GUI *)

ROUTINE Handle_GUI   (* structured text *)
   // Start and stop of ventilator
   
   HMI_ScreenNo :=0;
   
   If HMIStart then
   	Start_Stop :=1;
   	HMI_ScreenNo :=2;
   end_if;
   
   If HMIStop then
      Start_Stop :=0;
      HMI_ScreenNo :=1;
   End_if;
   
   
   if Start_Stop then									// If momantary push botton from GUI is on
   
   	if not VentOn then;								// If VentOn from ISR_ValveCtrl is NOT on
   		StartVent := 1;								// Set start signal to MainFlow sequence
   	end_if;
   
   else												// If stop from GUI
   
   	if VentOn then;									// If Ventilator is running in ISR_ValveCtrl
   		StopVent :=1;								// Set stop signal to MainFlow sequence
   	end_if;
   end_if;
   
   
   // Control of the F1 puch botton - Shifts between the 4 input just above the Fx bottons
   if data_changed then;								// start timer if data is changed
   	Timer := Timer+1;
   	if Timer >= 25 then;
   
   		TimerDone := 1;								// Set timer done
   		Timer := 0;
   	end_if;
   end_if;
   
   IF F1_pushed_new AND NOT F1_pushed_old Then
   	F1_pushed_old := 1;
   	IF F1_pushed_new THEN
   		IF data_changed THEN						// reset timer if data if changed repeatedly
   			data_changed := 0;
   			Timer := 0;								// reset timer
   
   		END_IF;
   		data_changed :=1;							// signal the timer to start
   		IF NOT(state_selected) THEN
   			state := last_state;
   			state_selected := 1;
   		ELSE
   			IF state <3 THEN
   			state := (state+1);
   			ELSE state := 0;
   		end_if;
   
   		END_IF;
   		CASE state OF
   			0: 	state0 := 1;
   				state1 := 0;
   				state2 := 0;
   				state3 := 0;
   			1: 	state0 := 0;
   				state1 := 1;
   				state2 := 0;
   				state3 := 0;
   			2: 	state0 := 0;
   				state1 := 0;
   				state2 := 1;
   				state3 := 0;
   			3: 	state0 := 0;
   				state1 := 0;
   				state2 := 0;
   				state3 := 1;
   		ELSE;
   		END_CASE;
   	END_If;
   END_IF;
   
   
   if not F1_pushed_new AND F1_pushed_old then;
   	F1_pushed_old :=0;
   end_if;
   
   
   // Control of the F2 botton - Add value to selected variable
   
   IF F2_pushed_new  AND NOT F2_pushed_old Then
   	F2_pushed_old := 1;
   	IF (F2_pushed_new AND state_selected) THEN			// increment value if state is selected
   		IF data_changed THEN							// reset timer if data if changed repeatedly
   			data_changed :=0;
   			Timer := 0;									// reset timer
   		END_IF;
   		data_changed := 1;								// signal the timer to start
   		CASE state OF
   			0:	FiO2	:= FiO2 + 5;				// increment value in case the O2 is selected
   				if FiO2 >= 100 then;
   					FiO2 := 100;
   				else;
   
   				end_if;
   			1:	Vt	:= Vt + 50;					// increment value in case the Vt is selected
   				if Vt >= 600 then;
   					Vt := 600;
   				else;
   
   				end_if;
   			2:	RRate 	:= RRate + 1;				// increment value in case the RRin is selected
   				if RRate >= 35 then;
   					RRate := 35;
   				else;
   
   				end_if;
   			3:	IE_counter := IE_counter + 1;		// increment value in case the I:E is selected
   				if IE_counter >= 2  then;
   					IE_counter := 2;
   
   				else;
   
   				end_if;
   				COP(IE[IE_counter], I_E, 82);
   		ELSE;
   		END_CASE;
   	END_IF;
   END_IF;
   
   if not F2_pushed_new AND F2_pushed_old then;
   	F2_pushed_old :=0;
   end_if;
   
   
   // Control of the F3 botton - Sub value to selected variable
   
   IF F3_pushed_new AND NOT F3_pushed_old Then
   	F3_pushed_old := 1;
   	IF (F3_pushed_new AND state_selected) THEN		// decrement value if state is selected
   		IF data_changed THEN						// reset timer if data if changed repeatedly
   			data_changed := 0;
   			Timer := 0;								// reset timer
   		END_IF;
   		data_changed := 1;							// signal the timer to start
   		CASE state OF
   			0:	FiO2 	:= FiO2 - 5;			// decrement value in case the O2 is selected
   				if FiO2 <= 0 then;
   					FiO2 := 0;
   				else;
   					//FiO2 := 0;
   				end_if;
   			1:	Vt	:= Vt - 50;				// decrement value in case the Vt is selected
   				if Vt <= 200 then;
   					Vt := 200;
   				else;
   
   				end_if;
   			2:	RRate 	:= RRate - 1;				// decrement value in case the RRin is selected
   				if RRate <= 6 then;
   					RRate := 6;
   				else;
   
   				end_if;
   			3:	IE_counter := IE_counter - 1;			// increment value in case the I:E is selected
   				if IE_counter <= 0  then;
   					IE_counter := 0;
   				//COP(IE[IE_counter], I_E, 82);
   				else;
   
   				end_if;
   				COP(IE[IE_counter], I_E, 82);
   		ELSE;
   		END_CASE;
   	END_IF;
   END_IF;
   
   if not F3_pushed_new AND F3_pushed_old then;
   	F3_pushed_old :=0;
   end_if;
   
   
   // If timer is done then deselect all states for new start
   
   IF TimerDone THEN
   	COP(Messages_to_user[0], message, 82);
   	data_changed := 0;
   	last_state := state;
   	state_selected := 0;
   	state0 := 0;
   	state1 := 0;
   	state2 := 0;
   	state3 := 0;
   	TimerDone := 0;
   ELSE
   	IF data_changed THEN
   		Time := Timer*200;
   		COP(Time, message, 82);
   		TimerDone :=0;
   	END_IF;
   END_IF;
   
   
   
   
END_ROUTINE
END_PROGRAM

PROGRAM initVent   (* main routine Main *)
VAR
   Oneshot : DINT;
END_VAR

ROUTINE Init_ISR_PressWatchID   (* structured text *)
   // Init of Pressure Watch
   // Routine only runs once
END_ROUTINE

ROUTINE initISR_ValveCtrl   (* structured text *)
   // Init of Valve Control
   // Routine only runs once
   
   // Fill BreathDurationArr with -1 only on first breath, for messuring average values
   AOI_FillArrayReal50(Fill50,BreathDurationArr, -1, 50);
   flowCalcOn := 0;		// No calculation of messurement - set to 1 if messurement ***** TEMP Soulution *****
   
   
END_ROUTINE

ROUTINE Main   (* structured text *)
   case StateInitVent of
   
   	10: 																// Prepare for transfer of data from calcBreath routine
   
   		COP(nextInspO2FlowCtrl[0], inspO2FlowCtrl[0], 650);				// Copy calculated data to running data
   		COP(nextInspAirFlowCtrl[0], inspAirFlowCtrl[0], 650);			// Copy calculated data to running data
   		COP(nextExpOpenCloseCtrl[0], expOpenCloseCtrl[0], 1000);		// Copy calculated data to running data
   		inspCountLength := nextInspCountLength;							// Copy lenght of inspiratory array calculated to runnung data
   		expCountLength := nextExpCountLength;							// Copy lenght of expiratory array calculated to runnung data
   
   		if inspCountLength >20 and expCountLength >20 then;				// Check values is correct
   			StateInitVent := 20;										// Set next stage
   		else
   			StartVent :=0;												// Stop ventilation
   			VentOn := 0; 												// Set do not run to ISR_ValveCtrl
   			COP(Messages_to_user[1], message, 82);						// Write to user that lenght insp or exp is not ok
   		end_if;
   
   
   	20:
   		JSR(initISR_ValveCtrl);											// Jump to init for ISR_ValveCtrl - only runs once
   		JSR(Init_ISR_PressWatchID);										// Jump to init for ISR_PressWatchID - only runs once
   
   		VentOn := 1; 													// Set start to ISR_ValveCtrl
   		StartVent := 0;													// Reset start bit
   		StateInitVent := 99;											// Set sequence finished state
   
   end_case;
END_ROUTINE
END_PROGRAM

PROGRAM ISR_ValveCtrl   (* main routine Main *)
VAR
   PressHtresholdUser : INT := 45;
   PressHtresholdUser1 : REAL := 35.0;
END_VAR

ROUTINE Main   (* structured text *)
   Pressure := 100.0/16000.0 * (AnalogInputPressure - 4000.0);
   //PressHtreshold := ((PressHtresholdUser1/100.0)*16000.0)+4000.0;
   
   
   // Control that either inspiratory or expiratory is set
   if (Insp and Exp) or (not Insp and not Exp) then;
   	if inspCount < inspCountLength and expCount < expCountLength then;
   		Exp := 1;											// Select expiatory
   		Insp := 0;											// Deselect inspiratory
   	end_if;
   	if inspCount < inspCountLength then;
   		Insp := 1;											// Select inspiraty
   		Exp := 0;											// DeSelect expiatory
   	end_if;
   	if expCount < expCountLength then;
   		Insp := 0;											// Deselect inspiratory
   		Exp := 1;											// Select expiatory
   	end_if;
   end_if;
   
   if VentOn then;
   
   	if StateValveCtrl = 0 then;
   
   		// Control if Inspiratory or expiatory
   		if Insp then;
   			StateValveCtrl :=10;								// Inspiratory
   			if _StartPosition <> _StartpositionOld then;
   				_StartPosition := counter;
   				_StartpositionOld := _StartPosition;
   			end_if;
   		end_if;
   
   		if Exp then
   			StateValveCtrl :=100;								// Expiatory
   		end_if;
   	End_if;
   
   	if StateValveCtrl = 10 then;
   		// Start of the Inspiratory
   		inspCount := inspCount +1;								// Count inspiratory up one in the cycle
   		expCount := 0;											// Reset expiatory counter
   		if Pressure > PressHtresholdUser1 then;							// Analog pressure High warning is high from input
   			StateValveCtrl := 11;								// Go to high pressure routine
   		else
   			StateValveCtrl := 20;								// Go to normal routine
   		end_if;
   	end_if;
   
   	if StateValveCtrl = 11 then;
   		// Close valves - high alarm on the Analog input will disapear when preassure is lower than high alarm
   		AnalogOutFlowO2 := 0;											// Close O2 valve
   		AnalogOutFlowAir := 0;											// Close Air Valve
   		expOpen :=1;											// Output - Open expiatory valve
   		StateValveCtrl := 30;									// Next state
   	end_if;
   
   	if StateValveCtrl = 20 then;
   		// Normal routine - set values to open valve
   		expOpen := 0;											// Output - close the expiatory valve
   		MCSV(GetSlaveValue, O2Up, inspO2FlowCtrl[inspCount], O2mAOut, O2mASlope, O2mADer);
   		AnalogOutFlowO2 := 1.03*O2mAOut;								// Set value to analog output control of O2
   		MCSV(GetSlaveValue, AirUp, inspAirFlowCtrl[inspCount], AirmAOut, AirmASlope, AirmADer);
   		AnalogOutFlowAir := 1.03*AirmAOut;							// Set value to analog output control of Air
   		StateValveCtrl := 30;									// Next state
   	end_if;
   
   	if StateValveCtrl = 30 then;
   		// Control if inspiratory has ended
   		if inspCount >= inspCountLength then;					// The Inspiratory has ended
   			Insp :=	0;											// Deselect inspiratory
   			Exp := 1;											// Select expiatory
   
   			if newInspFlowAvil then;							// New Inspiratory data is avalible
   				StateValveCtrl :=31;							// Set to new data for next cyclus is avalible
   			else
   				StateValveCtrl :=0;								// Start over
   			end_if;
   		else
   			StateValveCtrl :=0;									// Start over
   		end_if;
   	end_if;
   
   	if StateValveCtrl = 31 then;
   
   		COP(nextInspO2FlowCtrl[0], inspO2FlowCtrl[0], 650);		// Copy new O2 data to next inspiratory
   		COP(nextInspAirFlowCtrl[0], inspAirFlowCtrl[0], 650);	// Copy new Air data to next inspiratory
   		inspCountLength := nextInspCountLength;					// Copy new lenght of inspiratory
   		newInspFlowAvil := 0;									// Reset new Inspiratory data is avalible
   		StateValveCtrl := 0;									// Start over
   
   	end_if;
   
   	if StateValveCtrl = 100 then;
   		// Start of the Expiatory
   		expCount := expCount +1;									// Count expiratory up one in the cycle
   		inspCount := 0;												// Reset inspiratory counter
   		AnalogOutFlowO2 := 0;												// Close Inspiratory O2 valve
   		AnalogOutFlowAir := 0;												// Close Inspiratory Air valve
   		expOpen := expOpenCloseCtrl[expCount].0;					// Set state of expiratory valve
   
   		if expCount >= expCountLength then;
   			StateValveCtrl :=101;									// The Expiratory has ended
   			if _endPosition <> _endPositionOld then;
   				_endPosition := counter;
   				_endPositionOld := _endPosition;
   			end_if;
   		else
   			StateValveCtrl :=0;										// Start over
   		end_if;
   	end_if;
   
   	if StateValveCtrl = 101 then;
   		Insp :=1;													// Select inspiratory
   		Exp := 0; 													// DeSelect expiatory
   
   		if flowCalcOn then;
   
   			_StartPointBerfore := _StartPointBerfore;
   			_StartPosition:= _StartPosition;
   			_endPosition := _endPosition ;
   			_PointAfterEnd := _PointAfterEnd;
   
   
   			if (_endPosition -_StartPosition) + _StartPointBerfore +_PointAfterEnd < 999 then;
   
   				if _endPosition - _StartPosition > 0 then
   
   					StartSendPosition := _StartPosition - _StartPointBerfore;
   
   					if StartSendPosition < 0 then
   
   					_CopSource := 999 + StartSendPosition;
   					_CopLength := abs(StartSendPosition+1)*2;
   					COP(FlowAir[_CopSource,0],FlowArrMem[0,0],_CopLength);
   					COP(FlowO2[_CopSource,0],FlowO2Mem[0,0],_CopLength);
   					COP(PressArr[_CopSource,0],PressArrMem[0,0],_CopLength);
   
   					_CopSource1 := 0;
   					_CopDes1 := _CopLength + 1;
   					_CopLength1 := abs(StartSendPosition)+1;
   					COP(FlowAir[_CopSource1,0],FlowArrMem[_CopDes1 ,0],_CopLength1);
   					COP(FlowO2[_CopSource1,0],FlowO2Mem[_CopDes1 ,0],_CopLength1);
   					COP(PressArr[_CopSource1,0],PressArrMem[_CopDes1 ,0],_CopLength1);
   
   				else
   
   					_CopSource3 := StartSendPosition+1;
   					_CopLength3 :=_StartPointBerfore*2;
   					COP(FlowAir[_CopSource3,0],FlowArrMem[0,0],_CopLength3);
   					COP(FlowO2[_CopSource3,0],FlowO2Mem[0,0],_CopLength3);
   					COP(PressArr[_CopSource3,0],PressArrMem[0,0],_CopLength3);
   
   				end_if;
   
   				_EndSendPosition := _endPosition + _PointAfterEnd;
   
   				If _EndSendPosition > 999 then
   
   					_CopSource4 := _StartPosition + 1;
   					_CopDes4 := _StartPointBerfore;
   					_CopLength4 := ( 999 - _StartPosition + 1)*2;
   					COP(FlowAir[_CopSource4,0],FlowArrMem[_CopDes4,0],_CopLength4);
   					COP(FlowO2[_CopSource4,0],FlowO2Mem[_CopDes4,0],_CopLength4);
   					COP(PressArr[_CopSource4,0],PressArrMem[_CopDes4,0],_CopLength4);
   
   					_CopSource5 := 0;
   					_CopDes5 := _CopDes4 + 999 - _StartPosition;
   					_CopLength5 := (_EndSendPosition - 999) *2;
   					COP(FlowAir[_CopSource5,0],FlowArrMem[_CopDes5,0],_CopLength5);
   					COP(FlowO2[_CopSource5,0],FlowO2Mem[_CopDes5,0],_CopLength5);
   					COP(PressArr[_CopSource5,0],PressArrMem[_CopDes5,0],_CopLength5);
   
   				else
   
   					_CopSource6 := _StartPosition;
   					_CopDes6 := _StartPointBerfore;
   					_CopLength6 := (_EndSendPosition - _StartPosition) * 2;
   					COP(FlowAir[_CopSource6,0],FlowArrMem[_CopDes6,0],_CopLength6);
   					COP(FlowO2[_CopSource6,0],FlowO2Mem[_CopDes6,0],_CopLength6);
   					COP(PressArr[_CopSource6,0], PressArrMem[_CopDes6,0],_CopLength6);
   
   				End_if;
   
   				else
   
   					StartSendPosition := _StartPosition - _StartPointBerfore;
   					_CopSource7 := StartSendPosition;
   					_CopLength7 := (999 - StartSendPosition + 1) *2;
   					COP(FlowAir[_CopSource7,0],FlowArrMem[0,0],_CopLength7);
   					COP(FlowO2[_CopSource7,0],FlowO2Mem[0,0],_CopLength7);
   					COP(PressArr[_CopSource7,0], PressArrMem[0,0],_CopLength7);
   
   					_EndSendPosition := _endPosition + _PointAfterEnd;
   					_CopSource8 := 0;
   					_CopDes8 := (999 - StartSendPosition +1);
   					_CopLength8 := _EndSendPosition *2;
   					COP(FlowAir[_CopSource8,0],FlowArrMem[_CopDes8,0],_CopLength8);
   					COP(FlowO2[_CopSource8,0],FlowO2Mem[_CopDes8,0],_CopLength8);
   					COP(PressArr[_CopSource8,0], PressArrMem[_CopDes8,0],_CopLength8);
   
   				end_if;
   			end_if;
   
   			_endPositionOld :=0;
   			_StartpositionOld := 0;
   			CalcNewData := 1;
   
   		else
   
   		 CalcNewData := 0;
   
   		end_if;
   
   		if NewExpOpenCloseAvail then;								// New Expiatory data is avalible
   			StateValveCtrl := 102;									// Next state
   		else
   			StateValveCtrl := 0;									// Start over
   		end_if;
   	end_if;
   
   	if StateValveCtrl = 102 then;
   		COP(nextExpOpenCloseCtrl[0], expOpenCloseCtrl[0], 1000);	// Copy new close/open data to next expiatory
   		expCountLength := nextExpCountLength;						// Copy new lenght of expiatory
   		NewExpOpenCloseAvail := 0;									// Reset Expiatory data is avalible
   		StateValveCtrl := 0;										// Start over
   
   	end_if;
   end_if;
END_ROUTINE
END_PROGRAM

PROGRAM MainFlow   (* main routine Main *)

ROUTINE Main   (* structured text *)
   // Set MainFlow to start over
   if StateMain = 0 then;
   	StateMain := 10;
   end_if;
   
   IE_E := IE_counter +1;
   
   // see if new data is valible from GUI
   CsumData := FiO2+Vt + RRate + IE_I + IE_E + inspPauseTime + inspRampTime;
   
   If CsumData <> CsumDataOld then;
   	CsumDataOld := CsumData;
   	NewSettings :=1;
   	FiO2Running := FiO2;
   	VtRunning := Vt;
   	RRateRunning := RRate;
   	IE_IRunning := IE_I;
   	IE_ERunning := IE_E;
   	inspPauseTimeRunning := inspPauseTime;
   	inspRampTimeRunning := inspRampTime;
   end_if;
   
   
   
   // MainFlow sequence
   case StateMain of
   
   	// Run Setup
   	10: if SetupDone then;						// If setup is done
   			StateMain := 20;					// Set next stage
   			SetupState := 0;
   
   		else
   
   			if SetupState = 0 then;
   				SetupState := 10;
   			end_if;								// Start the setup program
   
   		end_if;
   
   	// Run CalcBreath
   	20:	if NewSettings then;					// If changes has happend on the GUI
   
   			if StateCalcBreath = 0 then;
   				StateCalcBreath := 10;				// Start the CalcBreath setup
   			end_if;
   		else
   			StateMain := 30;					// Set next stage
   		end_if;
   
   	// Stop Ventilation
   	30: if StopVent then;													// Stop ventilation
   			if Exp then
   				if expCount > (expCountLength - 20) then; 					// Stop ventilatio 20*scanrate befor expiratory ends
   					VentOn :=0 ;											// Stop ventilation routine
   					AOI_FillArray_Real2D(FillLoop,FlowAir,0,2000);				// Clear all raw data
   					AOI_FillArray_Real2D(FillLoop,FlowO2,0,2000);				// Clear all raw data
   					AOI_FillArray_Real2D(FillLoop,PressArr,0,2000);				// Clear all raw data
   					AOI_FillArray_Real2D(FillLoop,FlowArrMem,0,2000);			// Clear all raw data
   					AOI_FillArray_Real2D(FillLoop,FlowO2Mem ,0,2000);			// Clear all raw data
   					AOI_FillArray_Real2D(FillLoop,PressArrMem,0,2000);			// Clear all raw data
   					AOI_FillArray_Real2D(FillLoop,_edbFlowArrFiltered,0,2000);	// Clear all raw data
   					AOI_FillArray_Real2D(FillLoop,_edbFlowO2Filtered,0,2000);	// Clear all raw data
   					AOI_FillArray_Real2D(FillLoop,_edbPressArrFiltered,0,2000);	// Clear all raw data
   					StopVent := 0;											// Reset the stop command
   					Insp := 1;												// Select inspiratory next start first
   					Exp := 0;												// Deselect expiratory next start
   					expCount := 0;											// Reset the expiratory count
   					StateMain := 0;											// Reset sequence and start over
   
   				end_if;
   			end_if;
   		else
   			StateMain := 40;									// Set next stage
   		end_if;
   
   	// Run initVent
   	40:	if StartVent then;										// If ventilator is started
   
   			if StateInitVent = 0 then;
   				StateInitVent := 10;						// Start the initVent program
   			end_if;
   
   		else
   
   			StateMain := 0;
   			StateInitVent :=0;
   
   		end_if;
   
   end_case;
END_ROUTINE
END_PROGRAM

PROGRAM measArray   (* main routine Main *)
VAR
   Flow : REAL[1000,2];
END_VAR

ROUTINE FirstScan   (* structured text *)
   // From Analog_values
   
   counter :=0;
   SampelRateChangeAllowed := 0;
   Samplerate := 100 ;
   Samplerate_Old := 0;
   
   AOI_FillArray_Real2D(FillLoop,FlowAir,0,2000);
   AOI_FillArray_Real2D(FillLoop,PressArr,0,2000);
   //ClearArray_2D(FillLoop,FlowO2);		// Clear all raw data
   
   // Main flow
   
   StateMain := 10;
   SetupDone := 0;
   NewSettings := 1;
   StartVent := 0;
   StopVent := 0;
   VentOn := 0;
   
   // Setup
   
   SetupState := 0;
   
   
   // GUI
   
   data_changed :=0;
   
   
   // measCalc
   
   COP(RunModes[0], Mode, 82);	// Set Mode to 'VC'
   inspStartI := 0;
   inspPauseStartI := 0;
   expStartI := 0;
   expEndI := 0;
   totTime := 0;  //in s
   endI := 0;
   PplatBreathFrac := 0.2;
   
   AOI_FillArrayReal50(Fill50, PpeakArr, 0, 50);			//Float, 50 length array with Ppeak from measCalc(), used for minAvg
   AOI_FillArrayReal50(Fill50, PEEPArr, 0, 50);			//Float, 50 length array with positive end expiratory pressure in cmH2O, from measCalc()
   AOI_FillArrayReal50(Fill50, FlowImaxArr, 0, 50); 		//Float, 50 length array with max insp flow in l/min, from measCalc()
   AOI_FillArrayReal50(Fill50, PplatArr, 0, 50);			//Float, 50 length array with plateau insp pressure in cmH2O, from measCalc()
   AOI_FillArrayReal50(Fill50, RRArr, 0, 50);				//Float, 50 length array with respiratory rate in 1/min, from measCalc()
   AOI_FillArrayReal50(Fill50, VtiArr, 0, 50);				//Float, 50 length array with insp tidal volume in ml, from measCalc()
   AOI_FillArrayReal50(Fill50, MVArr, 0, 50);				//Float, 50 length array with minute ventilation in l/min, from measCalc()
   AOI_FillArrayReal50(Fill50, CrsDynArr, 0, 50);			//Float, 50 length array with dynamic respiraotry system compliance in ml/cmH2O, from measCalc()
   AOI_FillArrayReal50(Fill50, CrsQStatArr, 0, 50);		//Float, 50 length array with quasistatic respiratory system compliance in ml/cmH2O, from measCalc()
   AOI_FillArrayReal50(Fill50, RawArr, 0, 50); 			//Float, 50 length array with airway resistance in cmH2O/l/s, from measCalc()
   AOI_FillArrayReal50(Fill50, BreathDurationArr, 0, 50); 	//FLOAT, 50 length array with seconds for each breath for calculation of minute avgVentStateArr. Calculated from knowing meas at 100Hz for all breath data
   
   // CalcBreath
   
   StateCalcBreath := 0;		// Reset sequence
   valveUpdInterval := 10; 	//in ms Frequency 1000/10 = 100Hz
   maxFlowAllowed := 100; 		//In L/min. Sensor works until 830 ml/s (=49.8 l/min) Note: I will see if we have options to work around this as it will severely limit our options for settings
   
   // See if first time setup is done, the default values else presistent values from controller
   if FiO2 = 0 then;
   	FiO2 := 4;
   else
   	FiO2 := FiO2Running;
   end_if;
   
   if Vt = 0 then;
   	Vt := 350;
   else
   	Vt := VtRunning;
   end_if;
   
   if RRate = 0 then;
   	RRate := 15;
   else
   	RRate := RRateRunning;
   end_if;
   
   if IE_I = 0 then;
   	IE_I := 1;
   else
   	IE_I := IE_IRunning;
   end_if;
   
   if IE_E = 0 then;
   	IE_E := 2;
   else
   	IE_E := IE_ERunning;
   end_if;
   
   if inspPauseTime = 0 then;
   	inspPauseTime := 10;
   else
   	inspPauseTime := inspPauseTimeRunning;
   end_if;
   
   if inspRampTime = 0 then;
   	inspRampTime := 5;
   else
   	inspRampTime := inspRampTimeRunning;
   end_if;
   
   
   // Breath detect
   _StartPointBerfore := 30;
   _StartPosition:= 0;
   _endPosition := 0;
   _PointAfterEnd := 30;
   
END_ROUTINE

ROUTINE Main   (* structured text *)
   
   // If 1. scan in PLC
   if s:fs then;
   	jsr(FirstScan,0);
   end_if;
   
   // Jump to subroutine
   jsr(measArrays,0);
   
END_ROUTINE

ROUTINE measArrays   (* structured text *)
   // Enables to change scanrate
   // Special on a Rockwell PLC were you can change scan rates on the fly
   // Settings can be between 50hz or 100hz - alternativ it can be a fixed setting
   
   
   if Samplerate <> Samplerate_Old then;
   
   	if Samplerate <= 50 then;
   		Samplerate :=50;							// Set samplerate to 50 Hz if less is choosen
   	end_if;
   
   	if Samplerate > 100 then;
   		Samplerate := 100;							// Set samplerate to 100 Hz if higher is choosen
   	end_if;
   	TimeRate := (1000/Samplerate)*1000;				// Calc from Hz to ms
   	SSV(Task,P_Sample_p5,Rate,TimeRate);				// Shift sample rate on data collection
   	SSV(Task,P_Sample_p8,Rate,TimeRate);				// Shift sample rate on data collection
   	Samplerate_Old := Samplerate;					// Update parameter
   	GSV(Task,P_Sample_p5,Rate,NewTimeRate_p5);			// Get the time rate
   	GSV(Task,P_Sample_p8,Rate,NewTimeRate_p8);			// Get the time rate
   
   	if TimeRate = NewTimeRate_p5 and TimeRate = NewTimeRate_p8 then;
   		SampelRateChangeAllowed := 0;				// Stop change again
   		Samplerate_Old := 0;
   	end_if;
   end_if;
   
   
   
   // FIFO fill - load raw analog data into array
   if counter >= 0 and counter <= 999 then;								// Test counter values is between array values
   	Flow[counter,0] := (AnalogInputFlow*1)/1000;						// Write Total flow meassure into array 1. dimension
   	Flow[counter,0] := 0;												// Write data read into array 2. dimension
   	FlowAir[counter,0] := (AnalogInputFlowAir*75)/1000;					// Write flowAir meassure into array 1. dimension
   	FlowAir[counter,1] := 0;											// Write data read into array 2. dimension
   	FlowO2[counter,0] := (AnalogInputFlowO2*75)/1000;					// Write flowO2 meassure into array 1. dimension
   	FlowO2[counter,1] := 0;												// Write data read into array 2. dimension
   	PressArr[counter,0] := (AnalogInputPressure*6.37322633125)/1000 ;	// Write pressure meassure into array 1. dimension
   	PressArr[counter,1] := 0;											// Write data read into array 2. dimension
   
   	// ----------------------------------------------------------------------------
   	// -----------------------   C O D E    F R O M    E D B  ---------------------
   	//  All my variables start with _edb.
   	// Filtered values are stored in arrays:
   	//   _edbFlowArrFiltered
   	//   _edbFlowO2Filtered
   	//   _edbPressArrFiltered
   	// Note that initial setup of filters could be moved in a first scan
   	//   initialization routine (code between lines:
   	// *********************  Setup filters  ***************************
   	//   ...
   	// ******************  End of setup filters  ***********************
   	//
   	// I'm assuming here that all filter
       // are setup in the same way ( same window size, same type, ... ).
   	// In this isnt true the following code must be modified.
   
   	if counter = 0 then
   
   		// *********************  Setup filters  ****************************
   		// The lines in this section never change. Hence they could be moved
   		// in a first scan initialization.
   
   			// Set the window size of the filter.
   			// The total window size will be: 2 * _edbHalfWindowFilterSize + 1
   			// Maximum allowed value is 15
   			_edbHalfWindowFilterSize := 5; // To be defined
   
   
   			// Set the type of the filter.
   			// Mean filter (1) is basic a convolution and requires setting the
   			//   weights
   			_edbTypeOfFilter  := 0; // 0: MEDIAN; 1: MEAN
   			_edbParUseWeigths := 0; // Not used with a median filter
   
   			// In case _edbTypeOfFilter = 1 and _edbParUseWeigths := 1
   			// weights must be set.
   			// ...
   
   			// After having decided the above parameters, let's setup the
   			//   filters:
   			_edbAoiFilterFlowAir.Par_nWindowLeft   := _edbHalfWindowFilterSize;
   			_edbAoiFilterFlowAir.Par_nWindowsRight := _edbHalfWindowFilterSize;
   			_edbAoiFilterFlowAir.Par_eType         := _edbTypeOfFilter;
   			_edbAoiFilterFlowAir.Par_bUseWeights   := _edbParUseWeigths;
   
   			_edbAoiFilterFlowO2.Par_nWindowLeft   := _edbHalfWindowFilterSize;
   			_edbAoiFilterFlowO2.Par_nWindowsRight := _edbHalfWindowFilterSize;
   			_edbAoiFilterFlowO2.Par_eType         := _edbTypeOfFilter;
   			_edbAoiFilterFlowO2.Par_bUseWeights   := _edbParUseWeigths;
   
   			_edbAoiFilterPress.Par_nWindowLeft   := _edbHalfWindowFilterSize;
   			_edbAoiFilterPress.Par_nWindowsRight := _edbHalfWindowFilterSize;
   			_edbAoiFilterPress.Par_eType         := _edbTypeOfFilter;
   			_edbAoiFilterPress.Par_bUseWeights   := _edbParUseWeigths;
   		// ******************  End of setup filters  ************************
   
   		// ******************  Init filters' cycle  ************************
   		// The following lines must be execute when an acquisition cycle starts
   		//  (they cannot be moved in a first scan initialization routine)
   		_edbAoiFilterFlowAir.In_bInitialize := 1;
   		_edbAoiFilterFlowO2.In_bInitialize := 1;
   		_edbAoiFilterPress.In_bInitialize := 1;
   		// **************  End of init filters' cycle  *********************
   
   	end_if;
   
   	// Calculate filtered values
   	AOI_FilterSignal( _edbAoiFilterFlowAir, AnalogInputFlowAir, _edbParWeights );
   	AOI_FilterSignal( _edbAoiFilterPress, AnalogInputPressure, _edbParWeights );
   	AOI_FilterSignal( _edbAoiFilterFlowO2, AnalogInputFlowO2, _edbParWeights );
   
   	// Check if initial buffering has finished so we can start storing values.
   	// First _edbHalfWindowFilterSize elements of the array won't be calculated.
   	// Last _edbHalfWindowFilterSize elements of the array won't be calculated as well.
   	_edbCanStore := not _edbAoiFilterFlowAir.Out_Buffering and
   	                not _edbAoiFilterFlowO2.Out_Buffering  and
   					not _edbAoiFilterPress.Out_Buffering   and
   	                counter >= 2 * _edbHalfWindowFilterSize; // This last condition should be true when the previouos conditions are true.
   	if _edbCanStore then
   		_edbIdx := counter - _edbHalfWindowFilterSize; // Calculated filtered data is delayed by _edbHalfWindowFilterSize acquisitions
   		_edbFlowArrFiltered[_edbIdx,0] := _edbAoiFilterFlowAir.Out_rFilteredSignalDelayed;
   		_edbFlowArrFiltered[_edbIdx,1] := 0;
   		_edbFlowO2Filtered[_edbIdx,0] := _edbAoiFilterPress.Out_rFilteredSignalDelayed;
   		_edbFlowO2Filtered[_edbIdx,1] := 0;
   		_edbPressArrFiltered[_edbIdx,0] := _edbAoiFilterFlowO2.Out_rFilteredSignalDelayed;
   		_edbPressArrFiltered[_edbIdx,1] := 0;
   	end_if;
   	// ---------------  E N D    O F   C O D E    F R O M    E D B  ---------------
   	// ----------------------------------------------------------------------------
   
   	counter := counter +1;								// next count
   end_if;
   
   if counter >= 999 then;									// If count is at end of array
   	counter := 0;										// Reset counter
   end_if;
   
END_ROUTINE
END_PROGRAM
